{attribute addProperty BoxType "KL1408"}
{attribute addProperty Id "Channel_1Channel_70B606D100Channel_2Channel_70B606D100Channel_3Channel_70B606D100Channel_4Channel_70B606D100Channel_5Channel_70B606D100Channel_6Channel_70B606D100Channel_7Channel_70B606D100Channel_8Channel_70B606D100"}
{attribute addProperty CRC "2612289876"}
{attribute addProperty SizeInBites "0"}
{attribute addProperty SizeInBytes "0"}
TYPE KL1408_9BB46154 :
STRUCT
	{attribute addProperty Name "Channel_1"}
	Channel_1 : Channel_70B606D1;
	{attribute addProperty Name "Channel_2"}
	Channel_2 : Channel_70B606D1;
	{attribute addProperty Name "Channel_3"}
	Channel_3 : Channel_70B606D1;
	{attribute addProperty Name "Channel_4"}
	Channel_4 : Channel_70B606D1;
	{attribute addProperty Name "Channel_5"}
	Channel_5 : Channel_70B606D1;
	{attribute addProperty Name "Channel_6"}
	Channel_6 : Channel_70B606D1;
	{attribute addProperty Name "Channel_7"}
	Channel_7 : Channel_70B606D1;
	{attribute addProperty Name "Channel_8"}
	Channel_8 : Channel_70B606D1;
END_STRUCT
END_TYPE

(* stored: Version 1.2.0.0, ProductVersion 3.1.4024.9
   DUT KL1408_9BB46154: Id {5dd52853-1433-48ae-9958-cefef07dac66} *)
